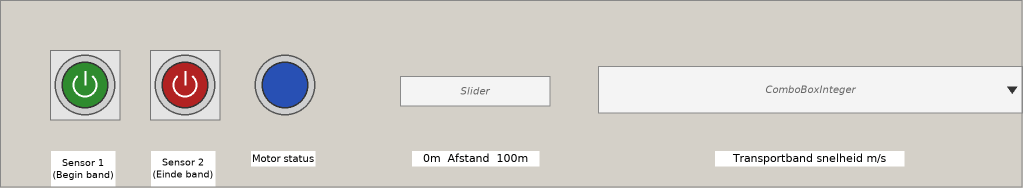
VISUALIZATION Visualization  // 1023x188
    Lamp1 (250,50 70x70), variable: GVL.MotorStatus, style: Lamp-Lamp1-Blue
    PowerSwitch (50,50 70x70), variable: GVL.ProductGedetecteerd1, behaviour: TOGGLE, style: Switch-PowerSwitch-Green
    PowerSwitch (150,50 70x70), variable: GVL.ProductGedetecteerd2, behaviour: TOGGLE, style: Switch-PowerSwitch-Red
    Slider (400,76 150x30), variable: GVL.Afstand, scale 0..100
    Textfield (50,150 66x38), "Sensor 1 (Begin band)"
    Textfield (150,150 66x37), "Sensor 2 (Einde band)"
    Textfield (250,150 66x17), "Motor status"
    Textfield (411,150 129x17), "0m Afstand 100m"
    ComboBoxInteger (598,66 425x47), variable: GVL.Snelheid
    Textfield (714,150 191x17), "Transportband snelheid m/s"
END_VISUALIZATION

(* stored: Version 1.1.0.1, ProductVersion 3.1.4024.12
   Visu Visualization: Id {84067154-05ff-47c7-9e48-17ec631654ff} *)
